TYPE
    ST_KeyValue : STRUCT
        ID  : STRING;
        Typ : STRING;
    END_STRUCT
END_TYPE

(* stored: Version 1.1.0.1
   DUT ST_KeyValue: Id {f5b3d48b-446b-4f31-aeff-db3c8130d9fc} *)
